// TIA Portal V20 export
FUNCTION_BLOCK "FB_Get_Out_Rework_Conveyor_Belt"   // FB8, LAD
{ S7_Optimized_Access := 'TRUE' }
// stored: AutoNumber false, MemoryReserve 100, SetENOAutomatically false
   VAR_INPUT
      Emergency_Stop_Release : Bool;
      Sensor_Water_Fountain_Geting_Exit_Rework_Conveyor_Belt : Bool;
      Button_Water_Fountain_Get_Exit_Rework_Conveyor_Belt : Bool;
      Sensor_Spinner_Entrace_Functional_Test_Position_Advanced : Bool;
      Sensor_Water_Fountain_Entrace_Functional_Test_Spinner_Conveyor_Belt : Bool;
   END_VAR
   VAR_OUTPUT
      Turn_On_Conveyor_Belt_Motor_Rework_Conveyor_Belt_Get_Entrace_Functional_Test : Bool;
   END_VAR
   VAR
      Aux_Trig_0 : Bool;
      Aux_Trig_1 : Bool;
      Aux_Trig_2 : Bool;
      Aux_Trig_3 : Bool;
      Aux_Trig_4 : Bool;
      Aux_Trig_5 : Bool;
      Aux_Trig_6 : Bool;
      Aux_Trig_7 : Bool;
      Button_Is_Pressed : Bool;
   END_VAR
BEGIN

REGION Network 1
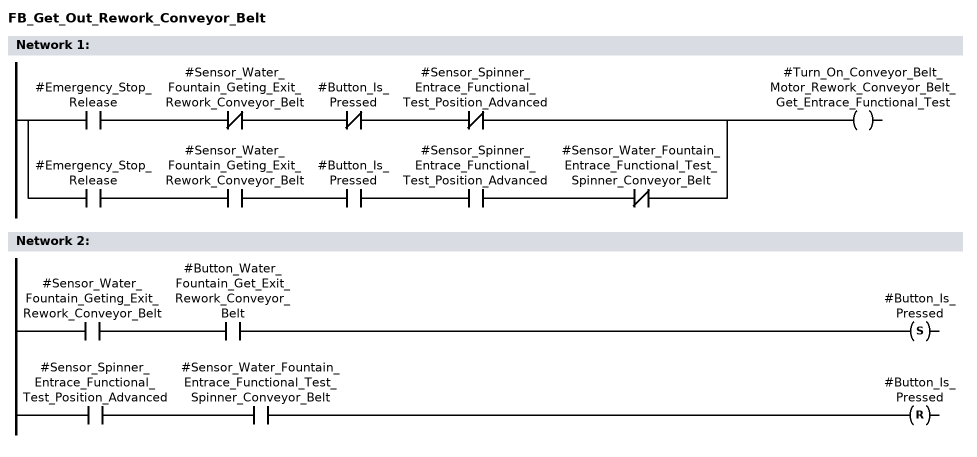
   RUNG wire#powerrail
      Contact( #Emergency_Stop_Release )
      I_Contact( #Sensor_Water_Fountain_Geting_Exit_Rework_Conveyor_Belt )
      I_Contact( #Button_Is_Pressed )
      I_Contact( #Sensor_Spinner_Entrace_Functional_Test_Position_Advanced )
      wire#w1
      Coil( #Turn_On_Conveyor_Belt_Motor_Rework_Conveyor_Belt_Get_Entrace_Functional_Test )
   END_RUNG
   RUNG wire#powerrail
      Contact( #Emergency_Stop_Release )
      Contact( #Sensor_Water_Fountain_Geting_Exit_Rework_Conveyor_Belt )
      Contact( #Button_Is_Pressed )
      Contact( #Sensor_Spinner_Entrace_Functional_Test_Position_Advanced )
      I_Contact( #Sensor_Water_Fountain_Entrace_Functional_Test_Spinner_Conveyor_Belt )
   END_RUNG wire#w1
   // the same network as SCL:
   #Turn_On_Conveyor_Belt_Motor_Rework_Conveyor_Belt_Get_Entrace_Functional_Test := (#Emergency_Stop_Release AND NOT #Sensor_Water_Fountain_Geting_Exit_Rework_Conveyor_Belt AND NOT #Button_Is_Pressed AND NOT #Sensor_Spinner_Entrace_Functional_Test_Position_Advanced) OR (#Emergency_Stop_Release AND #Sensor_Water_Fountain_Geting_Exit_Rework_Conveyor_Belt AND #Button_Is_Pressed AND #Sensor_Spinner_Entrace_Functional_Test_Position_Advanced AND NOT #Sensor_Water_Fountain_Entrace_Functional_Test_Spinner_Conveyor_Belt);
END_REGION

REGION Network 2
   RUNG wire#powerrail
      Contact( #Sensor_Water_Fountain_Geting_Exit_Rework_Conveyor_Belt )
      Contact( #Button_Water_Fountain_Get_Exit_Rework_Conveyor_Belt )
      S_Coil( #Button_Is_Pressed )
   END_RUNG
   RUNG wire#powerrail
      Contact( #Sensor_Spinner_Entrace_Functional_Test_Position_Advanced )
      Contact( #Sensor_Water_Fountain_Entrace_Functional_Test_Spinner_Conveyor_Belt )
      R_Coil( #Button_Is_Pressed )
   END_RUNG
   // the same network as SCL:
   IF #Sensor_Water_Fountain_Geting_Exit_Rework_Conveyor_Belt AND #Button_Water_Fountain_Get_Exit_Rework_Conveyor_Belt THEN
       #Button_Is_Pressed := TRUE;
   END_IF;
   IF #Sensor_Spinner_Entrace_Functional_Test_Position_Advanced AND #Sensor_Water_Fountain_Entrace_Functional_Test_Spinner_Conveyor_Belt THEN
       #Button_Is_Pressed := FALSE;
   END_IF;
END_REGION
END_FUNCTION_BLOCK
